// TIA Portal V19 program export: 2 tag tables, 0 data types, 4 data blocks, 2 code blocks (in call order from the OBs), 0 instance data blocks

VAR_GLOBAL   // PLC tag table "Default tag table"
   Tag_1 AT %M0.0 : Bool;
   Tag_2 AT %MW200 : Word;
   Tag_4 AT %M100.0 : Bool;
   Tag_5 AT %M100.1 : Bool;
END_VAR

VAR_GLOBAL   // PLC tag table "Default tag table_1"
   Tag_3 AT %M0.1 : Bool;
END_VAR

DATA_BLOCK "dataBlockGlobal"   // DB555
{ S7_Optimized_Access := 'TRUE' }
// stored: AutoNumber false, MemoryReserve 100
   VAR
      new : Array[0..99] of Byte;
   END_VAR
BEGIN
END_DATA_BLOCK

DATA_BLOCK "dataBlockLocal"   // DB111
{ S7_Optimized_Access := 'TRUE' }
// stored: AutoNumber false, MemoryReserve 100
BEGIN
END_DATA_BLOCK

DATA_BLOCK "next2DB"   // DB333
{ S7_Optimized_Access := 'TRUE' }
// stored: AutoNumber false, MemoryReserve 100
BEGIN
END_DATA_BLOCK

DATA_BLOCK "nextDB"   // DB222
{ S7_Optimized_Access := 'TRUE' }
// stored: AutoNumber false, MemoryReserve 100
   VAR
      data : Array[1..100] of Byte;
   END_VAR
BEGIN
END_DATA_BLOCK

ORGANIZATION_BLOCK "Main"   // OB1, LAD, ProgramCycle
TITLE = "Main Program Sweep (Cycle)"
{ S7_Optimized_Access := 'TRUE' }
// stored: SetENOAutomatically false
   VAR_INPUT
      Initial_Call : Bool;   // Initial call of this OB
      Remanence : Bool;   // =True, if remanent data are available
   END_VAR
   VAR_TEMP   // added for the SCL form of the ladder/FBD networks
      _w1 : Bool;
      _w2 : Bool;
   END_VAR
BEGIN

REGION Network 1
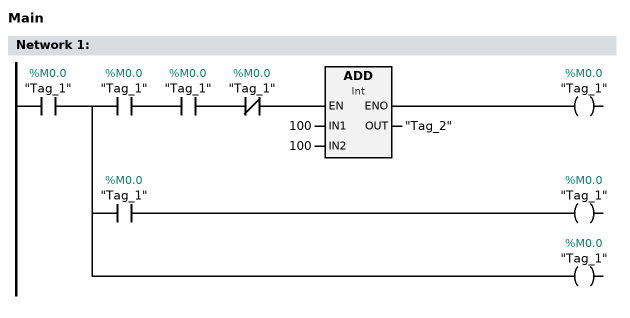
   RUNG wire#powerrail
      Contact( "Tag_1" )
      wire#w1
      Contact( "Tag_1" )
      Contact( "Tag_1" )
      I_Contact( "Tag_1" )
      { S7_Templates := "SrcType := Int" } Add(in1 := 100, in2 := 100, out => "Tag_2")
      Coil( "Tag_1" )
   END_RUNG
   RUNG wire#w1
      Contact( "Tag_1" )
      Coil( "Tag_1" )
   END_RUNG
   RUNG wire#w1
      Coil( "Tag_1" )
   END_RUNG
   // the same network as SCL:
   #_w1 := "Tag_1" AND "Tag_1" AND "Tag_1" AND NOT "Tag_1";
   IF #_w1 THEN "Tag_2" := 100 + 100; END_IF;
   #_w2 := "Tag_1";
   "Tag_1" := #_w1;
   "Tag_1" := #_w2 AND "Tag_1";
   "Tag_1" := #_w2;
END_REGION
END_ORGANIZATION_BLOCK

ORGANIZATION_BLOCK "Main_1"   // OB1000, LAD, ProgramCycle
TITLE = "Main Program Sweep (Cycle)"
// stored: AutoNumber false, SetENOAutomatically false
   VAR_INPUT
      Initial_Call : Bool;   // Initial call of this OB
      Remanence : Bool;   // =True, if remanent data are available
   END_VAR
BEGIN
END_ORGANIZATION_BLOCK
